ABB RAPID module: MotionProbe.mod

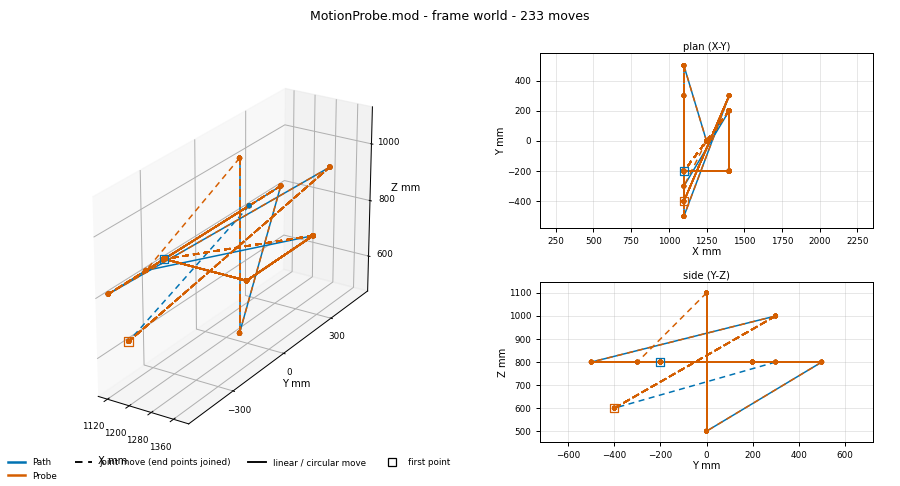
[picture p0: tool path of MotionProbe.mod in frame world, 233 of 233 moves have a stored position in this frame; points joined in program order, loops and branches not executed]
MODULE MotionProbe
    ! CrossArm - motion probe. In RobotStudio, PROC Probe times every run (ClkRead \HighRes) and
    ! writes 'name time' to HOME:/motionprobe.txt. PROC Path is what CrossArm converts. Real motion:
    ! RobotStudio only.
    CONST robtarget pCornerA:=[[1100,-200,800],[0,0.3826834,0.9238795,0],[-1,0,0,0],[9E+09,9E+09,9E+09,9E+09,9E+09,9E+09]];
    CONST robtarget pCornerB:=[[1400,-200,800],[0,0.3826834,0.9238795,0],[-1,0,0,0],[9E+09,9E+09,9E+09,9E+09,9E+09,9E+09]];
    CONST robtarget pCornerC:=[[1400,200,800],[0,0.3826834,0.9238795,0],[0,0,0,0],[9E+09,9E+09,9E+09,9E+09,9E+09,9E+09]];
    CONST robtarget pLineA:=[[1100,-300,800],[0,0.3826834,0.9238795,0],[-1,0,0,0],[9E+09,9E+09,9E+09,9E+09,9E+09,9E+09]];
    CONST robtarget pLineB:=[[1100,300,800],[0,0.3826834,0.9238795,0],[0,0,0,0],[9E+09,9E+09,9E+09,9E+09,9E+09,9E+09]];
    CONST robtarget pJointA:=[[1100,-400,600],[0,0.3826834,0.9238795,0],[-1,0,0,0],[9E+09,9E+09,9E+09,9E+09,9E+09,9E+09]];
    CONST robtarget pJointB:=[[1400,300,1000],[0,0.3826834,0.9238795,0],[0,0,0,0],[9E+09,9E+09,9E+09,9E+09,9E+09,9E+09]];
    CONST robtarget pSwingA:=[[1100,-500,800],[0,0.3826834,0.9238795,0],[-1,0,0,0],[9E+09,9E+09,9E+09,9E+09,9E+09,9E+09]];
    CONST robtarget pSwingB:=[[1100,500,800],[0,0.3826834,0.9238795,0],[0,0,0,0],[9E+09,9E+09,9E+09,9E+09,9E+09,9E+09]];
    CONST robtarget pRiseA:=[[1250,0,500],[0,0.3826834,0.9238795,0],[0,0,0,0],[9E+09,9E+09,9E+09,9E+09,9E+09,9E+09]];
    CONST robtarget pRiseB:=[[1250,0,1100],[0,0.3826834,0.9238795,0],[0,0,0,0],[9E+09,9E+09,9E+09,9E+09,9E+09,9E+09]];
    VAR clock clk;

    PROC Path()
        MoveL pCornerA,v1000,fine,tool0;
        MoveL pCornerB,v1000,fine,tool0;
        MoveL pCornerC,v1000,fine,tool0;
        MoveL pLineA,v1000,fine,tool0;
        MoveL pLineB,v1000,fine,tool0;
        MoveJ pJointA,v1000,fine,tool0;
        MoveJ pJointB,v1000,fine,tool0;
        MoveL pSwingA,v1000,fine,tool0;
        MoveL pSwingB,v1000,fine,tool0;
        MoveL pRiseA,v1000,fine,tool0;
        MoveL pRiseB,v1000,fine,tool0;
    ENDPROC

    PROC Probe()
        VAR iodev f;
        Open "HOME:" \File:="motionprobe.txt", f \Write;
        Close f;
        MoveJ pJointA,v1000,fine,tool0;
        ClkReset clk;
        ClkStart clk;
        MoveJ pJointB,v100,fine,tool0;
        WaitTime\InPos,0;
        ClkStop clk;
        Log "joint v100";
        MoveJ pJointA,v1000,fine,tool0;
        ClkReset clk;
        ClkStart clk;
        MoveJ pJointB,v200,fine,tool0;
        WaitTime\InPos,0;
        ClkStop clk;
        Log "joint v200";
        MoveJ pJointA,v1000,fine,tool0;
        ClkReset clk;
        ClkStart clk;
        MoveJ pJointB,v300,fine,tool0;
        WaitTime\InPos,0;
        ClkStop clk;
        Log "joint v300";
        MoveJ pJointA,v1000,fine,tool0;
        ClkReset clk;
        ClkStart clk;
        MoveJ pJointB,v500,fine,tool0;
        WaitTime\InPos,0;
        ClkStop clk;
        Log "joint v500";
        MoveJ pJointA,v1000,fine,tool0;
        ClkReset clk;
        ClkStart clk;
        MoveJ pJointB,v800,fine,tool0;
        WaitTime\InPos,0;
        ClkStop clk;
        Log "joint v800";
        MoveJ pJointA,v1000,fine,tool0;
        ClkReset clk;
        ClkStart clk;
        MoveJ pJointB,v1000,fine,tool0;
        WaitTime\InPos,0;
        ClkStop clk;
        Log "joint v1000";
        MoveJ pJointA,v1000,fine,tool0;
        ClkReset clk;
        ClkStart clk;
        MoveJ pJointB,v1500,fine,tool0;
        WaitTime\InPos,0;
        ClkStop clk;
        Log "joint v1500";
        MoveJ pJointA,v1000,fine,tool0;
        ClkReset clk;
        ClkStart clk;
        MoveJ pJointB,v2000,fine,tool0;
        WaitTime\InPos,0;
        ClkStop clk;
        Log "joint v2000";
        MoveJ pJointA,v1000,fine,tool0;
        ClkReset clk;
        ClkStart clk;
        MoveJ pJointB,v3000,fine,tool0;
        WaitTime\InPos,0;
        ClkStop clk;
        Log "joint v3000";
        MoveJ pJointA,v1000,fine,tool0;
        ClkReset clk;
        ClkStart clk;
        MoveJ pJointB,vmax,fine,tool0;
        WaitTime\InPos,0;
        ClkStop clk;
        Log "joint vmax";
        MoveJ pSwingA,v1000,fine,tool0;
        ClkReset clk;
        ClkStart clk;
        MoveJ pSwingB,v100,fine,tool0;
        WaitTime\InPos,0;
        ClkStop clk;
        Log "swing v100";
        MoveJ pSwingA,v1000,fine,tool0;
        ClkReset clk;
        ClkStart clk;
        MoveJ pSwingB,v200,fine,tool0;
        WaitTime\InPos,0;
        ClkStop clk;
        Log "swing v200";
        MoveJ pSwingA,v1000,fine,tool0;
        ClkReset clk;
        ClkStart clk;
        MoveJ pSwingB,v300,fine,tool0;
        WaitTime\InPos,0;
        ClkStop clk;
        Log "swing v300";
        MoveJ pSwingA,v1000,fine,tool0;
        ClkReset clk;
        ClkStart clk;
        MoveJ pSwingB,v500,fine,tool0;
        WaitTime\InPos,0;
        ClkStop clk;
        Log "swing v500";
        MoveJ pSwingA,v1000,fine,tool0;
        ClkReset clk;
        ClkStart clk;
        MoveJ pSwingB,v800,fine,tool0;
        WaitTime\InPos,0;
        ClkStop clk;
        Log "swing v800";
        MoveJ pSwingA,v1000,fine,tool0;
        ClkReset clk;
        ClkStart clk;
        MoveJ pSwingB,v1000,fine,tool0;
        WaitTime\InPos,0;
        ClkStop clk;
        Log "swing v1000";
        MoveJ pSwingA,v1000,fine,tool0;
        ClkReset clk;
        ClkStart clk;
        MoveJ pSwingB,v1500,fine,tool0;
        WaitTime\InPos,0;
        ClkStop clk;
        Log "swing v1500";
        MoveJ pSwingA,v1000,fine,tool0;
        ClkReset clk;
        ClkStart clk;
        MoveJ pSwingB,v2000,fine,tool0;
        WaitTime\InPos,0;
        ClkStop clk;
        Log "swing v2000";
        MoveJ pSwingA,v1000,fine,tool0;
        ClkReset clk;
        ClkStart clk;
        MoveJ pSwingB,v3000,fine,tool0;
        WaitTime\InPos,0;
        ClkStop clk;
        Log "swing v3000";
        MoveJ pSwingA,v1000,fine,tool0;
        ClkReset clk;
        ClkStart clk;
        MoveJ pSwingB,vmax,fine,tool0;
        WaitTime\InPos,0;
        ClkStop clk;
        Log "swing vmax";
        MoveJ pRiseA,v1000,fine,tool0;
        ClkReset clk;
        ClkStart clk;
        MoveJ pRiseB,v100,fine,tool0;
        WaitTime\InPos,0;
        ClkStop clk;
        Log "rise v100";
        MoveJ pRiseA,v1000,fine,tool0;
        ClkReset clk;
        ClkStart clk;
        MoveJ pRiseB,v200,fine,tool0;
        WaitTime\InPos,0;
        ClkStop clk;
        Log "rise v200";
        MoveJ pRiseA,v1000,fine,tool0;
        ClkReset clk;
        ClkStart clk;
        MoveJ pRiseB,v300,fine,tool0;
        WaitTime\InPos,0;
        ClkStop clk;
        Log "rise v300";
        MoveJ pRiseA,v1000,fine,tool0;
        ClkReset clk;
        ClkStart clk;
        MoveJ pRiseB,v500,fine,tool0;
        WaitTime\InPos,0;
        ClkStop clk;
        Log "rise v500";
        MoveJ pRiseA,v1000,fine,tool0;
        ClkReset clk;
        ClkStart clk;
        MoveJ pRiseB,v800,fine,tool0;
        WaitTime\InPos,0;
        ClkStop clk;
        Log "rise v800";
        MoveJ pRiseA,v1000,fine,tool0;
        ClkReset clk;
        ClkStart clk;
        MoveJ pRiseB,v1000,fine,tool0;
        WaitTime\InPos,0;
        ClkStop clk;
        Log "rise v1000";
        MoveJ pRiseA,v1000,fine,tool0;
        ClkReset clk;
        ClkStart clk;
        MoveJ pRiseB,v1500,fine,tool0;
        WaitTime\InPos,0;
        ClkStop clk;
        Log "rise v1500";
        MoveJ pRiseA,v1000,fine,tool0;
        ClkReset clk;
        ClkStart clk;
        MoveJ pRiseB,v2000,fine,tool0;
        WaitTime\InPos,0;
        ClkStop clk;
        Log "rise v2000";
        MoveJ pRiseA,v1000,fine,tool0;
        ClkReset clk;
        ClkStart clk;
        MoveJ pRiseB,v3000,fine,tool0;
        WaitTime\InPos,0;
        ClkStop clk;
        Log "rise v3000";
        MoveJ pRiseA,v1000,fine,tool0;
        ClkReset clk;
        ClkStart clk;
        MoveJ pRiseB,vmax,fine,tool0;
        WaitTime\InPos,0;
        ClkStop clk;
        Log "rise vmax";
        MoveJ pLineA,v1000,fine,tool0;
        ClkReset clk;
        ClkStart clk;
        MoveL pLineB,v100,fine,tool0;
        WaitTime\InPos,0;
        ClkStop clk;
        Log "linear v100";
        MoveJ pLineA,v1000,fine,tool0;
        ClkReset clk;
        ClkStart clk;
        MoveL pLineB,v200,fine,tool0;
        WaitTime\InPos,0;
        ClkStop clk;
        Log "linear v200";
        MoveJ pLineA,v1000,fine,tool0;
        ClkReset clk;
        ClkStart clk;
        MoveL pLineB,v500,fine,tool0;
        WaitTime\InPos,0;
        ClkStop clk;
        Log "linear v500";
        MoveJ pLineA,v1000,fine,tool0;
        ClkReset clk;
        ClkStart clk;
        MoveL pLineB,v1000,fine,tool0;
        WaitTime\InPos,0;
        ClkStop clk;
        Log "linear v1000";
        MoveJ pLineA,v1000,fine,tool0;
        ClkReset clk;
        ClkStart clk;
        MoveL pLineB,v1500,fine,tool0;
        WaitTime\InPos,0;
        ClkStop clk;
        Log "linear v1500";
        MoveJ pLineA,v1000,fine,tool0;
        ClkReset clk;
        ClkStart clk;
        MoveL pLineB,v2000,fine,tool0;
        WaitTime\InPos,0;
        ClkStop clk;
        Log "linear v2000";
        MoveJ pCornerA,v1000,fine,tool0;
        ClkReset clk;
        ClkStart clk;
        MoveL pCornerB,v200,fine,tool0;
        MoveL pCornerC,v200,fine,tool0;
        WaitTime\InPos,0;
        ClkStop clk;
        Log "corner v200 fine";
        MoveJ pCornerA,v1000,fine,tool0;
        ClkReset clk;
        ClkStart clk;
        MoveL pCornerB,v200,z1,tool0;
        MoveL pCornerC,v200,fine,tool0;
        WaitTime\InPos,0;
        ClkStop clk;
        Log "corner v200 z1";
        MoveJ pCornerA,v1000,fine,tool0;
        ClkReset clk;
        ClkStart clk;
        MoveL pCornerB,v200,z5,tool0;
        MoveL pCornerC,v200,fine,tool0;
        WaitTime\InPos,0;
        ClkStop clk;
        Log "corner v200 z5";
        MoveJ pCornerA,v1000,fine,tool0;
        ClkReset clk;
        ClkStart clk;
        MoveL pCornerB,v200,z10,tool0;
        MoveL pCornerC,v200,fine,tool0;
        WaitTime\InPos,0;
        ClkStop clk;
        Log "corner v200 z10";
        MoveJ pCornerA,v1000,fine,tool0;
        ClkReset clk;
        ClkStart clk;
        MoveL pCornerB,v200,z20,tool0;
        MoveL pCornerC,v200,fine,tool0;
        WaitTime\InPos,0;
        ClkStop clk;
        Log "corner v200 z20";
        MoveJ pCornerA,v1000,fine,tool0;
        ClkReset clk;
        ClkStart clk;
        MoveL pCornerB,v200,z30,tool0;
        MoveL pCornerC,v200,fine,tool0;
        WaitTime\InPos,0;
        ClkStop clk;
        Log "corner v200 z30";
        MoveJ pCornerA,v1000,fine,tool0;
        ClkReset clk;
        ClkStart clk;
        MoveL pCornerB,v200,z50,tool0;
        MoveL pCornerC,v200,fine,tool0;
        WaitTime\InPos,0;
        ClkStop clk;
        Log "corner v200 z50";
        MoveJ pCornerA,v1000,fine,tool0;
        ClkReset clk;
        ClkStart clk;
        MoveL pCornerB,v200,z100,tool0;
        MoveL pCornerC,v200,fine,tool0;
        WaitTime\InPos,0;
        ClkStop clk;
        Log "corner v200 z100";
        MoveJ pCornerA,v1000,fine,tool0;
        ClkReset clk;
        ClkStart clk;
        MoveL pCornerB,v200,z150,tool0;
        MoveL pCornerC,v200,fine,tool0;
        WaitTime\InPos,0;
        ClkStop clk;
        Log "corner v200 z150";
        MoveJ pCornerA,v1000,fine,tool0;
        ClkReset clk;
        ClkStart clk;
        MoveL pCornerB,v200,z200,tool0;
        MoveL pCornerC,v200,fine,tool0;
        WaitTime\InPos,0;
        ClkStop clk;
        Log "corner v200 z200";
        MoveJ pCornerA,v1000,fine,tool0;
        ClkReset clk;
        ClkStart clk;
        MoveL pCornerB,v500,fine,tool0;
        MoveL pCornerC,v500,fine,tool0;
        WaitTime\InPos,0;
        ClkStop clk;
        Log "corner v500 fine";
        MoveJ pCornerA,v1000,fine,tool0;
        ClkReset clk;
        ClkStart clk;
        MoveL pCornerB,v500,z1,tool0;
        MoveL pCornerC,v500,fine,tool0;
        WaitTime\InPos,0;
        ClkStop clk;
        Log "corner v500 z1";
        MoveJ pCornerA,v1000,fine,tool0;
        ClkReset clk;
        ClkStart clk;
        MoveL pCornerB,v500,z5,tool0;
        MoveL pCornerC,v500,fine,tool0;
        WaitTime\InPos,0;
        ClkStop clk;
        Log "corner v500 z5";
        MoveJ pCornerA,v1000,fine,tool0;
        ClkReset clk;
        ClkStart clk;
        MoveL pCornerB,v500,z10,tool0;
        MoveL pCornerC,v500,fine,tool0;
        WaitTime\InPos,0;
        ClkStop clk;
        Log "corner v500 z10";
        MoveJ pCornerA,v1000,fine,tool0;
        ClkReset clk;
        ClkStart clk;
        MoveL pCornerB,v500,z20,tool0;
        MoveL pCornerC,v500,fine,tool0;
        WaitTime\InPos,0;
        ClkStop clk;
        Log "corner v500 z20";
        MoveJ pCornerA,v1000,fine,tool0;
        ClkReset clk;
        ClkStart clk;
        MoveL pCornerB,v500,z30,tool0;
        MoveL pCornerC,v500,fine,tool0;
        WaitTime\InPos,0;
        ClkStop clk;
        Log "corner v500 z30";
        MoveJ pCornerA,v1000,fine,tool0;
        ClkReset clk;
        ClkStart clk;
        MoveL pCornerB,v500,z50,tool0;
        MoveL pCornerC,v500,fine,tool0;
        WaitTime\InPos,0;
        ClkStop clk;
        Log "corner v500 z50";
        MoveJ pCornerA,v1000,fine,tool0;
        ClkReset clk;
        ClkStart clk;
        MoveL pCornerB,v500,z100,tool0;
        MoveL pCornerC,v500,fine,tool0;
        WaitTime\InPos,0;
        ClkStop clk;
        Log "corner v500 z100";
        MoveJ pCornerA,v1000,fine,tool0;
        ClkReset clk;
        ClkStart clk;
        MoveL pCornerB,v500,z150,tool0;
        MoveL pCornerC,v500,fine,tool0;
        WaitTime\InPos,0;
        ClkStop clk;
        Log "corner v500 z150";
        MoveJ pCornerA,v1000,fine,tool0;
        ClkReset clk;
        ClkStart clk;
        MoveL pCornerB,v500,z200,tool0;
        MoveL pCornerC,v500,fine,tool0;
        WaitTime\InPos,0;
        ClkStop clk;
        Log "corner v500 z200";
        MoveJ pCornerA,v1000,fine,tool0;
        ClkReset clk;
        ClkStart clk;
        MoveL pCornerB,v1000,fine,tool0;
        MoveL pCornerC,v1000,fine,tool0;
        WaitTime\InPos,0;
        ClkStop clk;
        Log "corner v1000 fine";
        MoveJ pCornerA,v1000,fine,tool0;
        ClkReset clk;
        ClkStart clk;
        MoveL pCornerB,v1000,z1,tool0;
        MoveL pCornerC,v1000,fine,tool0;
        WaitTime\InPos,0;
        ClkStop clk;
        Log "corner v1000 z1";
        MoveJ pCornerA,v1000,fine,tool0;
        ClkReset clk;
        ClkStart clk;
        MoveL pCornerB,v1000,z5,tool0;
        MoveL pCornerC,v1000,fine,tool0;
        WaitTime\InPos,0;
        ClkStop clk;
        Log "corner v1000 z5";
        MoveJ pCornerA,v1000,fine,tool0;
        ClkReset clk;
        ClkStart clk;
        MoveL pCornerB,v1000,z10,tool0;
        MoveL pCornerC,v1000,fine,tool0;
        WaitTime\InPos,0;
        ClkStop clk;
        Log "corner v1000 z10";
        MoveJ pCornerA,v1000,fine,tool0;
        ClkReset clk;
        ClkStart clk;
        MoveL pCornerB,v1000,z20,tool0;
        MoveL pCornerC,v1000,fine,tool0;
        WaitTime\InPos,0;
        ClkStop clk;
        Log "corner v1000 z20";
        MoveJ pCornerA,v1000,fine,tool0;
        ClkReset clk;
        ClkStart clk;
        MoveL pCornerB,v1000,z30,tool0;
        MoveL pCornerC,v1000,fine,tool0;
        WaitTime\InPos,0;
        ClkStop clk;
        Log "corner v1000 z30";
        MoveJ pCornerA,v1000,fine,tool0;
        ClkReset clk;
        ClkStart clk;
        MoveL pCornerB,v1000,z50,tool0;
        MoveL pCornerC,v1000,fine,tool0;
        WaitTime\InPos,0;
        ClkStop clk;
        Log "corner v1000 z50";
        MoveJ pCornerA,v1000,fine,tool0;
        ClkReset clk;
        ClkStart clk;
        MoveL pCornerB,v1000,z100,tool0;
        MoveL pCornerC,v1000,fine,tool0;
        WaitTime\InPos,0;
        ClkStop clk;
        Log "corner v1000 z100";
        MoveJ pCornerA,v1000,fine,tool0;
        ClkReset clk;
        ClkStart clk;
        MoveL pCornerB,v1000,z150,tool0;
        MoveL pCornerC,v1000,fine,tool0;
        WaitTime\InPos,0;
        ClkStop clk;
        Log "corner v1000 z150";
        MoveJ pCornerA,v1000,fine,tool0;
        ClkReset clk;
        ClkStart clk;
        MoveL pCornerB,v1000,z200,tool0;
        MoveL pCornerC,v1000,fine,tool0;
        WaitTime\InPos,0;
        ClkStop clk;
        Log "corner v1000 z200";
        MoveJ pCornerA,v1000,fine,tool0;
        ClkReset clk;
        ClkStart clk;
        MoveJ pCornerB,v500,fine,tool0;
        MoveJ pCornerC,v500,fine,tool0;
        WaitTime\InPos,0;
        ClkStop clk;
        Log "jcorner v500 fine";
        MoveJ pCornerA,v1000,fine,tool0;
        ClkReset clk;
        ClkStart clk;
        MoveJ pCornerB,v500,z1,tool0;
        MoveJ pCornerC,v500,fine,tool0;
        WaitTime\InPos,0;
        ClkStop clk;
        Log "jcorner v500 z1";
        MoveJ pCornerA,v1000,fine,tool0;
        ClkReset clk;
        ClkStart clk;
        MoveJ pCornerB,v500,z5,tool0;
        MoveJ pCornerC,v500,fine,tool0;
        WaitTime\InPos,0;
        ClkStop clk;
        Log "jcorner v500 z5";
        MoveJ pCornerA,v1000,fine,tool0;
        ClkReset clk;
        ClkStart clk;
        MoveJ pCornerB,v500,z10,tool0;
        MoveJ pCornerC,v500,fine,tool0;
        WaitTime\InPos,0;
        ClkStop clk;
        Log "jcorner v500 z10";
        MoveJ pCornerA,v1000,fine,tool0;
        ClkReset clk;
        ClkStart clk;
        MoveJ pCornerB,v500,z20,tool0;
        MoveJ pCornerC,v500,fine,tool0;
        WaitTime\InPos,0;
        ClkStop clk;
        Log "jcorner v500 z20";
        MoveJ pCornerA,v1000,fine,tool0;
        ClkReset clk;
        ClkStart clk;
        MoveJ pCornerB,v500,z30,tool0;
        MoveJ pCornerC,v500,fine,tool0;
        WaitTime\InPos,0;
        ClkStop clk;
        Log "jcorner v500 z30";
        MoveJ pCornerA,v1000,fine,tool0;
        ClkReset clk;
        ClkStart clk;
        MoveJ pCornerB,v500,z50,tool0;
        MoveJ pCornerC,v500,fine,tool0;
        WaitTime\InPos,0;
        ClkStop clk;
        Log "jcorner v500 z50";
        MoveJ pCornerA,v1000,fine,tool0;
        ClkReset clk;
        ClkStart clk;
        MoveJ pCornerB,v500,z100,tool0;
        MoveJ pCornerC,v500,fine,tool0;
        WaitTime\InPos,0;
        ClkStop clk;
        Log "jcorner v500 z100";
        MoveJ pCornerA,v1000,fine,tool0;
        ClkReset clk;
        ClkStart clk;
        MoveJ pCornerB,v500,z150,tool0;
        MoveJ pCornerC,v500,fine,tool0;
        WaitTime\InPos,0;
        ClkStop clk;
        Log "jcorner v500 z150";
        MoveJ pCornerA,v1000,fine,tool0;
        ClkReset clk;
        ClkStart clk;
        MoveJ pCornerB,v500,z200,tool0;
        MoveJ pCornerC,v500,fine,tool0;
        WaitTime\InPos,0;
        ClkStop clk;
        Log "jcorner v500 z200";
        MoveJ pCornerA,v1000,fine,tool0;
        ClkReset clk;
        ClkStart clk;
        MoveJ pCornerB,v1000,fine,tool0;
        MoveJ pCornerC,v1000,fine,tool0;
        WaitTime\InPos,0;
        ClkStop clk;
        Log "jcorner v1000 fine";
        MoveJ pCornerA,v1000,fine,tool0;
        ClkReset clk;
        ClkStart clk;
        MoveJ pCornerB,v1000,z1,tool0;
        MoveJ pCornerC,v1000,fine,tool0;
        WaitTime\InPos,0;
        ClkStop clk;
        Log "jcorner v1000 z1";
        MoveJ pCornerA,v1000,fine,tool0;
        ClkReset clk;
        ClkStart clk;
        MoveJ pCornerB,v1000,z5,tool0;
        MoveJ pCornerC,v1000,fine,tool0;
        WaitTime\InPos,0;
        ClkStop clk;
        Log "jcorner v1000 z5";
        MoveJ pCornerA,v1000,fine,tool0;
        ClkReset clk;
        ClkStart clk;
        MoveJ pCornerB,v1000,z10,tool0;
        MoveJ pCornerC,v1000,fine,tool0;
        WaitTime\InPos,0;
        ClkStop clk;
        Log "jcorner v1000 z10";
        MoveJ pCornerA,v1000,fine,tool0;
        ClkReset clk;
        ClkStart clk;
        MoveJ pCornerB,v1000,z20,tool0;
        MoveJ pCornerC,v1000,fine,tool0;
        WaitTime\InPos,0;
        ClkStop clk;
        Log "jcorner v1000 z20";
        MoveJ pCornerA,v1000,fine,tool0;
        ClkReset clk;
        ClkStart clk;
        MoveJ pCornerB,v1000,z30,tool0;
        MoveJ pCornerC,v1000,fine,tool0;
        WaitTime\InPos,0;
        ClkStop clk;
        Log "jcorner v1000 z30";
        MoveJ pCornerA,v1000,fine,tool0;
        ClkReset clk;
        ClkStart clk;
        MoveJ pCornerB,v1000,z50,tool0;
        MoveJ pCornerC,v1000,fine,tool0;
        WaitTime\InPos,0;
        ClkStop clk;
        Log "jcorner v1000 z50";
        MoveJ pCornerA,v1000,fine,tool0;
        ClkReset clk;
        ClkStart clk;
        MoveJ pCornerB,v1000,z100,tool0;
        MoveJ pCornerC,v1000,fine,tool0;
        WaitTime\InPos,0;
        ClkStop clk;
        Log "jcorner v1000 z100";
        MoveJ pCornerA,v1000,fine,tool0;
        ClkReset clk;
        ClkStart clk;
        MoveJ pCornerB,v1000,z150,tool0;
        MoveJ pCornerC,v1000,fine,tool0;
        WaitTime\InPos,0;
        ClkStop clk;
        Log "jcorner v1000 z150";
        MoveJ pCornerA,v1000,fine,tool0;
        ClkReset clk;
        ClkStart clk;
        MoveJ pCornerB,v1000,z200,tool0;
        MoveJ pCornerC,v1000,fine,tool0;
        WaitTime\InPos,0;
        ClkStop clk;
        Log "jcorner v1000 z200";
        TPWrite "motionprobe.txt written in HOME:";
    ENDPROC

    PROC Log(string name)
        VAR iodev f;
        Open "HOME:" \File:="motionprobe.txt", f \Append;
        Write f, name+" "+NumToStr(ClkRead(clk\HighRes),3);
        Close f;
    ENDPROC
ENDMODULE
